FUNCTION_BLOCK ContactorNO
VAR
	output AT %Q* : BOOL;
END_VAR

METHOD Close
VAR_INPUT
END_VAR
output := TRUE;
END_METHOD

PROPERTY IsClosed : BOOL
GET
IsClosed := output;
END_GET
END_PROPERTY

PROPERTY IsOpen : BOOL
GET
IsOpen := NOT output;
END_GET
END_PROPERTY

METHOD Open
VAR_INPUT
END_VAR
output := FALSE;
END_METHOD

END_FUNCTION_BLOCK

(* stored: Version 1.1.0.1, ProductVersion 3.1.4024.12
   POU ContactorNO: Id {2cbc9b42-ed95-4499-ad75-c76cb1ff34f7}, SpecialFunc None
   Method Close: Id {45ceba98-10de-4d40-81eb-8bf49e4e83a8}
   Property IsClosed: Id {ace5800f-0eee-4e61-8b2b-a5a26202c429}
   Get Get: Id {d5af05ec-0857-4b64-9d9b-1078ca905116}
   Property IsOpen: Id {de4f1fae-f444-44e6-b5c7-c0c86b30509a}
   Get Get: Id {29a8cf54-8a94-4e28-ab17-0655aae8c4dd}
   Method Open: Id {e843bc73-797c-4f41-8c7e-9b985c691d2f} *)
